FUNCTION_BLOCK ObjectDetect (* Template for a simple Basic Function Block Type *)
  (* Standard: 61499-2 *)
  (* Version 1.0, 2019-06-07, Promok *)
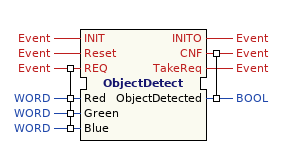
  EVENT_INPUT
    INIT;
    Reset;
    REQ WITH Red, Green, Blue; (* Normal Execution Request *)
  END_EVENT
  EVENT_OUTPUT
    INITO;
    CNF WITH ObjectDetected;
    TakeReq;
  END_EVENT
  VAR_INPUT
    Red : WORD; (* Input event qualifier *)
    Green : WORD;
    Blue : WORD;
  END_VAR
  VAR_OUTPUT
    ObjectDetected : BOOL;
  END_VAR
  VAR
    ObjectRecognized : BOOL; (* Internal Variable *)
    ReqAlreadyStarted : BOOL; (* Internal Variable *)
    StartRequest : BOOL; (* Internal Variable *)
    Init : BOOL; (* Internal Variable *)
    NewObject : BOOL; (* Internal Variable *)
  END_VAR
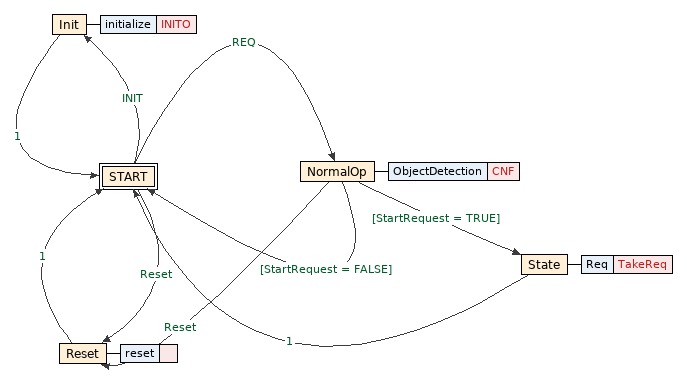
  EC_STATES
    START; (* Initial State *)
    NormalOp : ObjectDetection -> CNF; (* Normal execution *)
    Init : initialize -> INITO;
    Reset : reset;
    State : Req -> TakeReq;
  END_STATES
  EC_TRANSITIONS
    START TO NormalOp := REQ;
    Init TO START := 1;
    START TO Reset := Reset;
    Reset TO START := 1;
    NormalOp TO State := [StartRequest = TRUE];
    NormalOp TO START := [StartRequest = FALSE];
    State TO START := 1;
    NormalOp TO Reset := Reset;
    START TO Init := INIT;
  END_TRANSITIONS
  ALGORITHM ObjectDetection IN ST: (* new algorithm *)
IF Red>= 10 AND  Green >=20 AND Blue >=20 THEN
	IF Init = TRUE THEN
		NewObject := FALSE;
	END_IF;
	ObjectDetected := TRUE;

	IF ReqAlreadyStarted = FALSE AND NewObject = TRUE THEN
		StartRequest := TRUE;
	END_IF;

ELSE
		ObjectDetected := FALSE;
		NewObject := TRUE;
END_IF;

Init := FALSE;
  END_ALGORITHM
  ALGORITHM initialize IN ST: (* new algorithm *)
Init := TRUE;
NewObject := TRUE;
  END_ALGORITHM
  ALGORITHM reset IN ST: (* new algorithm *)
ReqAlreadyStarted := FALSE;
StartRequest := FALSE;
NewObject := TRUE;
Init := TRUE;
  END_ALGORITHM
  ALGORITHM Req IN ST: (* new algorithm *)
//ColourAlreadyDetected := TRUE;
ReqAlreadyStarted := TRUE;
StartRequest := FALSE;
NewObject := TRUE;
Init := TRUE;
  END_ALGORITHM
END_FUNCTION_BLOCK
